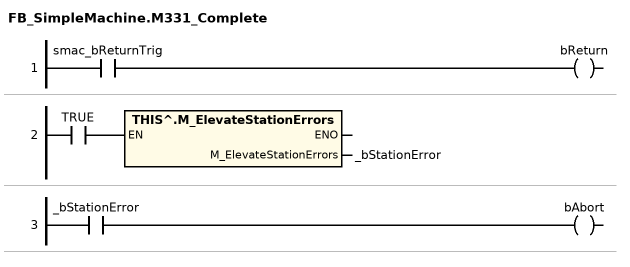
// NETWORK 1
bReturn := smac_bReturnTrig;

// NETWORK 2
_bStationError := THIS^.M_ElevateStationErrors();

// NETWORK 3
bAbort := _bStationError;
END_METHOD

(* In this state the most recent execution status should be maintained while
awaiting an explicit 'Unhold' command once internal conditions are satisfactory. *)
METHOD M411_Held : BOOL
VAR_OUTPUT
	(* This should be set to true if an explicit 'Unhold' command is received.
	Once set to true, the state machine will move to the 'Unholding' state. *)
	bUnhold	: BOOL;
	(* This should be set to true if an external source requests that the module
	exit its current state and come to a controlled stop. Once set to true, the
	state machine will move to the 'Stopping' state. *)
	bStop	: BOOL;
	(* This should be set to true if a potentially hazardous error or a safety
	fault has occurred in any tasks. Once set to true, the state machine will
	move to the 'Aborting' state. *)
	bAbort	: BOOL;
END_VAR
VAR
	_bStationError: BOOL;
END_VAR
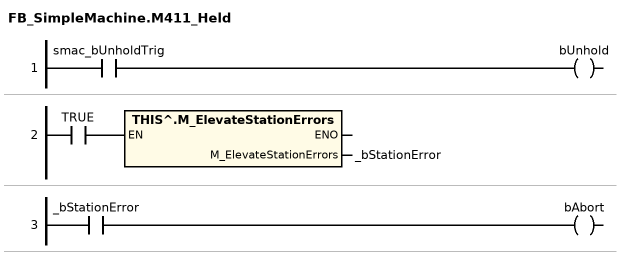
// NETWORK 1
bUnhold := smac_bUnholdTrig;

// NETWORK 2
_bStationError := THIS^.M_ElevateStationErrors();

// NETWORK 3
bAbort := _bStationError;
END_METHOD

(* In this state the most recent execution status should be maintained while
awaiting an explicit 'Unsuspend' command once external conditions are satisfactory. *)
METHOD M511_Suspended : BOOL
VAR_OUTPUT
	(* This should be set to true if an explicit 'Unsuspend' command is received.
	Once set to true, the state machine will move to the 'Unsuspending' state. *)
	bUnsuspend	: BOOL;
	(* This should be set to true if an external source requests that the module
	exit its current state and come to a controlled stop. Once set to true, the
	state machine will move to the 'Stopping' state. *)
	bStop	: BOOL;
	(* This should be set to true if a potentially hazardous error or a safety
	fault has occurred in any tasks. Once set to true, the state machine will
	move to the 'Aborting' state. *)
	bAbort	: BOOL;
END_VAR
VAR
	_bStationError: BOOL;
END_VAR
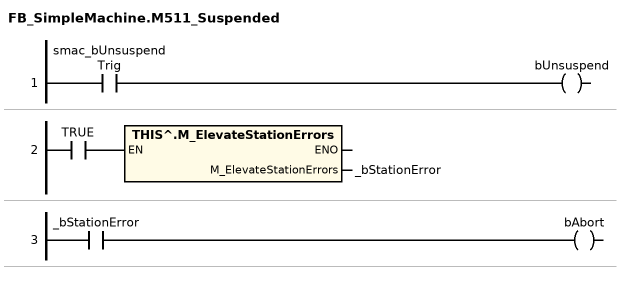
// NETWORK 1
bUnsuspend := smac_bUnsuspendTrig;

// NETWORK 2
_bStationError := THIS^.M_ElevateStationErrors();

// NETWORK 3
bAbort := _bStationError;
END_METHOD

END_FUNCTION_BLOCK

// Interfaces/State Machine/Stateful/I_ExecuteStateOnly
(* This interface only implements the methods for the Execute state. *)
INTERFACE I_ExecuteStateOnly EXTENDS I_SimpleExecuteStateOnly

(* Runs for a single cycle when entering the execute state. *)
METHOD M310_Execute_Entry : BOOL
VAR_INPUT
END_VAR
END_METHOD

(* Runs for a single cycle when exiting the execute state. *)
METHOD M312_Execute_Exit : BOOL
VAR_INPUT
END_VAR
END_METHOD

END_INTERFACE

// Interfaces/State Machine/Stateful/I_TransitionStatesOnly
(* This interface implements only the PackML transition states. *)
INTERFACE I_TransitionStatesOnly EXTENDS I_SimpleTransitionStatesOnly

(* Runs for a single cycle when entering the aborting state. *)
METHOD M000_Aborting_Entry : BOOL
VAR_INPUT
END_VAR
END_METHOD

(* Runs for a single cycle when exiting the aborting state. *)
METHOD M002_Aborting_Exit : BOOL
VAR_INPUT
END_VAR
END_METHOD

(* Runs for a single cycle when entering the clearing state. *)
METHOD M020_Clearing_Entry : BOOL
VAR_INPUT
END_VAR
END_METHOD

(* Runs for a single cycle when exiting the clearing state. *)
METHOD M022_Clearing_Exit : BOOL
VAR_INPUT
END_VAR
END_METHOD

(* Runs for a single cycle when entering the stopping state. *)
METHOD M100_Stopping_Entry : BOOL
VAR_INPUT
END_VAR
END_METHOD

(* Runs for a single cycle when exiting the stopping state. *)
METHOD M102_Stopping_Exit : BOOL
VAR_INPUT
END_VAR
END_METHOD

(* Runs for a single cycle when entering the resetting state. *)
METHOD M200_Resetting_Entry : BOOL
VAR_INPUT
END_VAR
END_METHOD

(* Runs for a single cycle when exiting the resetting state. *)
METHOD M202_Resetting_Exit : BOOL
VAR_INPUT
END_VAR
END_METHOD

(* Runs for a single cycle when entering the starting state. *)
METHOD M300_Starting_Entry : BOOL
VAR_INPUT
END_VAR
END_METHOD

(* Runs for a single cycle when exiting the starting state. *)
METHOD M302_Starting_Exit : BOOL
VAR_INPUT
END_VAR
END_METHOD

(* Runs for a single cycle when entering the completing state. *)
METHOD M320_Completing_Entry : BOOL
VAR_INPUT
END_VAR
END_METHOD

(* Runs for a single cycle when exiting the completing state. *)
METHOD M322_Completing_Exit : BOOL
VAR_INPUT
END_VAR
END_METHOD

(* Runs for a single cycle when entering the holding state. *)
METHOD M400_Holding_Entry : BOOL
VAR_INPUT
END_VAR
END_METHOD

(* Runs for a single cycle when exiting the holding state. *)
METHOD M402_Holding_Exit : BOOL
VAR_INPUT
END_VAR
END_METHOD

(* Runs for a single cycle when entering the unholding state. *)
METHOD M420_Unholding_Entry : BOOL
VAR_INPUT
END_VAR
END_METHOD

(* Runs for a single cycle when exiting the unholding state. *)
METHOD M422_Unholding_Exit : BOOL
VAR_INPUT
END_VAR
END_METHOD

(* Runs for a single cycle when entering the suspending state. *)
METHOD M500_Suspending_Entry : BOOL
VAR_INPUT
END_VAR
END_METHOD

(* Runs for a single cycle when exiting the suspending state. *)
METHOD M502_Suspending_Exit : BOOL
VAR_INPUT
END_VAR
END_METHOD

(* Runs for a single cycle when entering the unsuspending state. *)
METHOD M520_Unsuspending_Entry : BOOL
VAR_INPUT
END_VAR
END_METHOD

(* Runs for a single cycle when exiting the unsuspending state. *)
METHOD M522_Unsuspending_Exit : BOOL
VAR_INPUT
END_VAR
END_METHOD

END_INTERFACE

// Interfaces/Stations/I_StationDeviceControl
INTERFACE I_StationDeviceControl

(* Aborts all devices set in the station. *)
METHOD M_AbortDevices : BOOL
VAR_INPUT
END_VAR
END_METHOD

(* Clears all devices set in the station. *)
METHOD M_ClearDevices : BOOL
VAR_INPUT
END_VAR
END_METHOD

(* Completes all devices set in the station. *)
METHOD M_CompleteDevices : BOOL
VAR_INPUT
END_VAR
END_METHOD

(* Holds all devices set in the station. *)
METHOD M_HoldDevices : BOOL
VAR_INPUT
END_VAR
END_METHOD

(* Resets all devices set in the station. *)
METHOD M_ResetDevices : BOOL
VAR_INPUT
END_VAR
END_METHOD

(* Starts all devices set in the station. *)
METHOD M_StartDevices : BOOL
VAR_INPUT
END_VAR
END_METHOD

(* Stops all devices set in the station. *)
METHOD M_StopDevices : BOOL
VAR_INPUT
END_VAR
END_METHOD

(* Suspends all devices set in the station. *)
METHOD M_SuspendDevices : BOOL
VAR_INPUT
END_VAR
END_METHOD

(* Unholds all devices set in the station. *)
METHOD M_UnholdDevices : BOOL
VAR_INPUT
END_VAR
END_METHOD

(* Unsuspends all devices set in the station. *)
METHOD M_UnsuspendDevices : BOOL
VAR_INPUT
END_VAR
END_METHOD

END_INTERFACE

// Project Information/F_GetCompany
// This function has been automatically generated from the project information.
{attribute 'signature_flag' := '1073741824'}
{attribute 'TcGenerated'}
{attribute 'no-analysis'}
FUNCTION F_GetCompany : WSTRING
VAR_INPUT
	
END_VAR

F_GetCompany := "Sensata Technologies";

END_FUNCTION

// Project Information/F_GetTitle
// This function has been automatically generated from the project information.
{attribute 'signature_flag' := '1073741824'}
{attribute 'TcGenerated'}
{attribute 'no-analysis'}
FUNCTION F_GetTitle : WSTRING
VAR_INPUT
	
END_VAR

F_GetTitle := "Sensata_Common";

END_FUNCTION

// Project Information/F_GetVersion
// This function has been automatically generated from the project information.
{attribute 'signature_flag' := '1073741824'}
{attribute 'TcGenerated'}
{attribute 'no-analysis'}
FUNCTION F_GetVersion : ST_LibVersion
VAR_INPUT
	
END_VAR

F_GetVersion.iMajor := 1;
F_GetVersion.iMinor := 0;
F_GetVersion.iBuild := 0;
F_GetVersion.iRevision := 0;

END_FUNCTION
